# EPICS autosave request: iocBoot/iocJenaNV100D/auto_settings.req
file "JenaNV100D.req", P=$(P), R=$(R)
file "JenaNV100D_settings.req", P=$(P), R=$(R)
